Fanuc KAREL source: kd00046.KL

PROGRAM KD00046
%STACKSIZE=65535
%PRIORITY=65535
%NOLOCKGROUP
VAR
I : INTEGER
J : INTEGER
B : BOOLEAN
R : REAL
S : STRING[80]
-- UNRESOLVED DECLARATIONS (source type spelling not recovered)
-- V : TYPE_0x0013 (type_u16=0x0013)
BEGIN
-- UNSAFE_SOURCE_IR line 12: field_offset(V,0) = 1065353216
-- UNRESOLVED_PC line 13 opcodes [01 49 0A 82 0B] marker_code=20
END KD00046
